// TIA Portal V19 export
TYPE "Prod_Interruzioni"
   STRUCT
      STOP_FineTurno : Bool;
      STOP_FineTurno_Done : Bool;
      STOP_ControlloQualita : Bool;
      STOP_ControlloQualita_Done : Bool;
      O_ACT : Struct
         MES_IDP { ExternalWritable := 'False'} : String[30];
         Halted_Cause { ExternalWritable := 'False'} : "Prod_Halted_Str";
         Last_Halted_Cause_Code { ExternalWritable := 'False'; S7_SetPoint := 'True'} : Int;
         Mem_STOP : Bool;
      END_STRUCT;
      O_ENDING : Array[1.."PROD_ENDING_ITEMS"] of Struct
         MES_IDP { ExternalWritable := 'False'} : String[30];
         Halted_Cause { ExternalWritable := 'False'} : "Prod_Halted_Str";
         Last_Halted_Cause_Code { ExternalWritable := 'False'; S7_SetPoint := 'True'} : Int;
         Stopped_MEM : Int;
      END_STRUCT;
   END_STRUCT;
END_TYPE
